// TIA Portal V16 export
// export: Created 2022-11-17T15:49:02.6894183Z, ExportSetting WithDefaults, DisplayName Totally Integrated Automation Portal, DisplayVersion V16 Update 6, DisplayName TIA Portal Version Control Interface, DisplayVersion V16 Update 2, DisplayName TIA Portal Openness, DisplayVersion V16 Update 6, DisplayName SINAMICS Startdrive Advanced, DisplayVersion V16 Update 5, DisplayName SINAMICS Startdrive G130, G150, S120, S150, SINAMICS MV, S210, DisplayVersion V16 Update 5, DisplayName SINAMICS Startdrive G110M, G120, G120C, G120D, G120P, G115D, DisplayVersion V16 Update 5, DisplayName STEP 7 Professional, DisplayVersion V16 Update 6, DisplayName STEP 7 Safety, DisplayVersion V16, DisplayName WinCC Advanced, DisplayVersion V16 Update 6
FUNCTION_BLOCK "Inverter_Process_Data"   // FB1, FBD
{ S7_Optimized_Access := 'TRUE' }
VERSION : 0.1
// stored: AutoNumber false, IsIECCheckEnabled false, IsRetainMemResEnabled false, MemoryReserve 100, SetENOAutomatically false, UDAEnableTagReadback false
   VAR_INPUT
      control_word : Word := 16#0000;
      setpoint : Real;
      RD_address : HW_SUBMODULE;
      WR_address : HW_SUBMODULE;
      ref_quantity : Struct
         speed_p2000 : Real := 1500.0;
         current_p2002 : Real := 0.65;
         torque_p2003 : Real := 1.7;
      END_STRUCT;
   END_VAR
   VAR_OUTPUT
      status_word : Word;
      actual_speed : Real;
      actual_current : Real;
      actual_torque : Real;
      actual_alarm : Word;
      actual_fault : Word;
      RETVAL_RD : Word;
      RETVAL_WR : Word;
   END_VAR
   VAR_TEMP
      InData : Array[1..6] of Word;
      OutData : Array[1..6] of Word;
      actual_speed_INT : Int;
      actual_current_INT : Int;
      actual_torque_INT : Int;
      setpoint_INT : Int;
   END_VAR
BEGIN

REGION Network 1
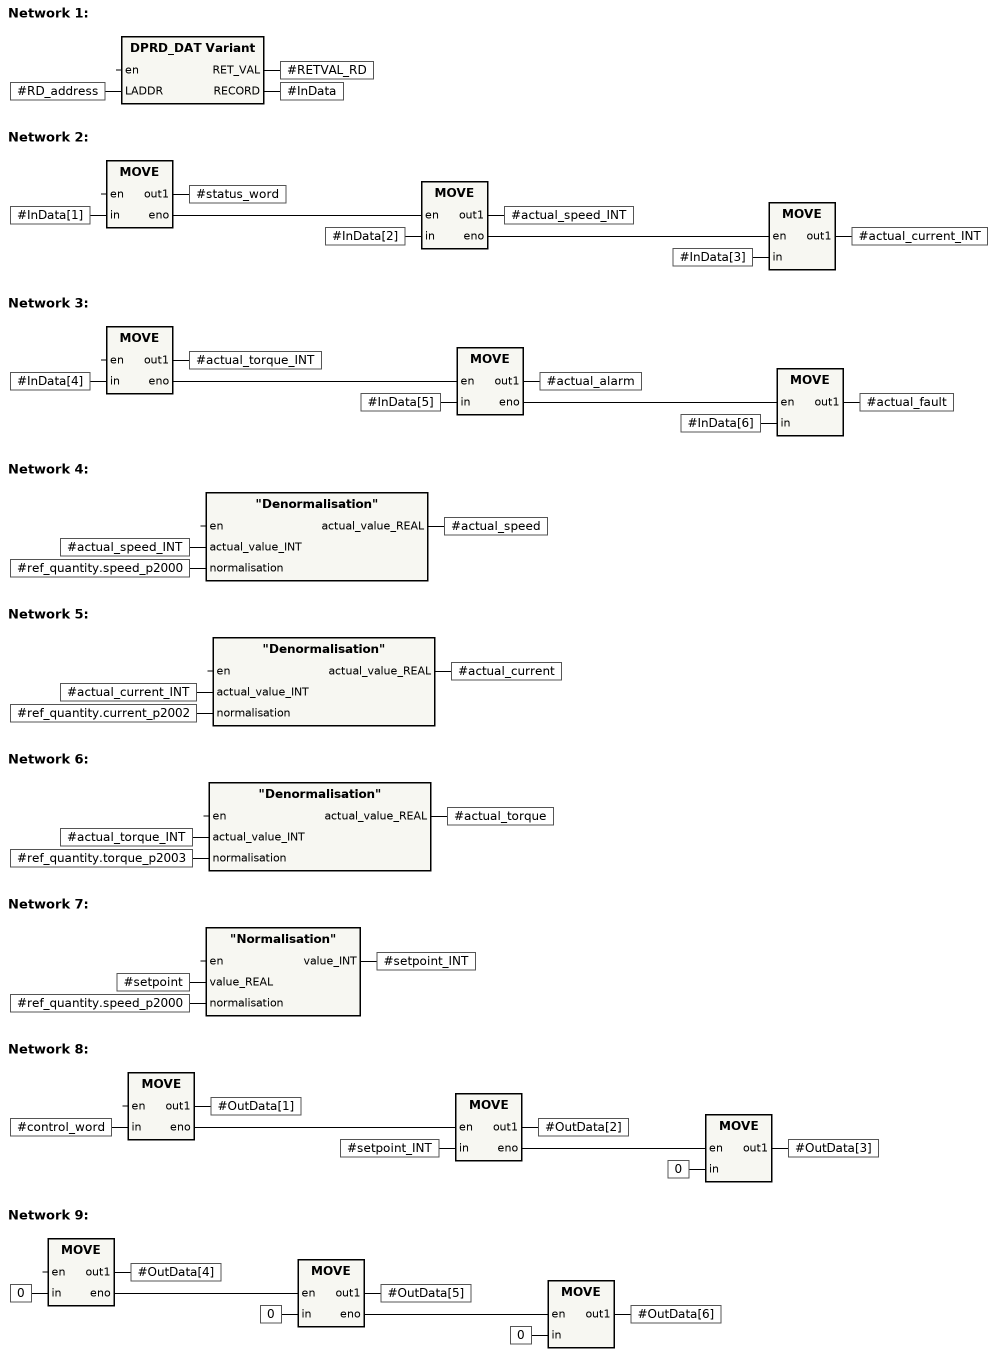
   #RETVAL_RD := DPRD_DAT(LADDR := #RD_address, RECORD => #InData);
END_REGION

REGION Network 2
   // ENO of a box is taken as its EN; it also drops when the box reports an error
   #status_word := #InData[1];
   #actual_speed_INT := #InData[2];
   #actual_current_INT := #InData[3];
END_REGION

REGION Network 3
   // ENO of a box is taken as its EN; it also drops when the box reports an error
   #actual_torque_INT := #InData[4];
   #actual_alarm := #InData[5];
   #actual_fault := #InData[6];
END_REGION

REGION Network 4
   "Denormalisation"(actual_value_INT := #actual_speed_INT,
                     normalisation := #ref_quantity.speed_p2000,
                     actual_value_REAL => #actual_speed);
END_REGION

REGION Network 5
   "Denormalisation"(actual_value_INT := #actual_current_INT,
                     normalisation := #ref_quantity.current_p2002,
                     actual_value_REAL => #actual_current);
END_REGION

REGION Network 6
   "Denormalisation"(actual_value_INT := #actual_torque_INT,
                     normalisation := #ref_quantity.torque_p2003,
                     actual_value_REAL => #actual_torque);
END_REGION

REGION Network 7
   "Normalisation"(value_REAL := #setpoint,
                   normalisation := #ref_quantity.speed_p2000,
                   value_INT => #setpoint_INT);
END_REGION

REGION Network 8
   // ENO of a box is taken as its EN; it also drops when the box reports an error
   #OutData[1] := #control_word;
   #OutData[2] := #setpoint_INT;
   #OutData[3] := 0;
END_REGION

REGION Network 9
   // ENO of a box is taken as its EN; it also drops when the box reports an error
   #OutData[4] := 0;
   #OutData[5] := 0;
   #OutData[6] := 0;
END_REGION

REGION Network 10
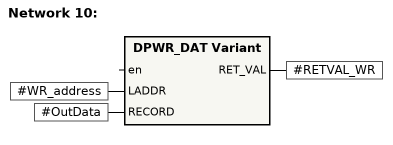
   #RETVAL_WR := DPWR_DAT(LADDR := #WR_address, RECORD := #OutData);
END_REGION
END_FUNCTION_BLOCK
